// Block: PPrgArchive15

DATA_BLOCK PPrgArchive15
VERSION : 0.1
   NON_RETAIN
   VAR
      PRG : Array[1401..1500] of PPrg_Data;
   END_VAR

BEGIN
   // No initialization required
END_DATA_BLOCK
